(*********************************** G.D S.p.A. - Technical Department ***********************************
============= PROGRAM INFO ============
FOLDER:             TBD
MACHINES INVOLVED:  TBD 

============= DESCRIPTION =============
csp main interface program

============= REVISIONS ===============
Date		Version	 	Author      	Description             
----------	-------		------------  	--------------------------------------------
2019/09/27 	0000.00	 	M.Grasso		Creation of the PRG

**********************************************************************************************************)
PROGRAM _csp_transfer_main_lowest
VAR
END_VAR

(*MAIN*)

	(*Brand*)
	
	(*Drives*)
	
	(*Motorization*)
	
	(*Cam Manager*)
	
	(*Services*)
	
	(*Interface*)
	
	(*Safety*)
	;

END_PROGRAM

(* stored: Version 1.1.0.1, ProductVersion 3.1.4022.12
   POU _csp_transfer_main_lowest: Id {e5e55cf1-dcd5-415c-8559-58130ec32b6f}, SpecialFunc None *)
